// TIA Portal V18 export
// export: Created 2026-03-12T16:04:35.7521041Z, ExportSetting WithDefaults, DisplayName Totally Integrated Automation Portal, DisplayVersion V18 Update 5, DisplayName TIA Portal Openness, DisplayVersion V18 Update 5, DisplayName TIA Portal Version Control Interface, DisplayVersion V18, DisplayName SINAMICS Startdrive Advanced, DisplayVersion V18, DisplayName SINAMICS Startdrive G130, G150, S120, S150, SINAMICS MV, S210, DisplayVersion V18, DisplayName SINAMICS Startdrive G110M, G120, G120C, G120D, G120P, G115D, DisplayVersion V18, DisplayName STEP 7 Professional, DisplayVersion V18 Update 5, DisplayName STEP 7 Safety, DisplayVersion V18, DisplayName WinCC Professional, DisplayVersion V18 Update 5
FUNCTION_BLOCK "FB_MOVE_SKID_DESARENADOR"   // FB33, SCL
{ S7_Optimized_Access := 'TRUE' }
VERSION : 0.1
// stored: AutoNumber true, IsIECCheckEnabled false, IsRetainMemResEnabled false, MemoryReserve 100, SetENOAutomatically false, UDAEnableTagReadback false
   VAR_INPUT
      Dados_Word : Array[10..64] of Int;
      Dados_Bool : Array[0..152] of Bool;
   END_VAR
   VAR_IN_OUT
      SKID_DESARENADOR : Struct
         EMERGENCIA_LIBERADA : Bool;
         AUTOMATICO : Bool;
         MANUAL : Bool;
         POSIÇÃO_INICLA_MANUAL : Bool;
         FLAG_BOMBA_01_LIGADA : Bool;
         FLAG_BOMBA_02_LIGADA : Bool;
         FLAG_SOBRECARGA_DESLOCAMENTO : Bool;
         FLAG_SOBRECARGA_ARRASTADOR01 : Bool;
         FLAG_SOBRECARGA_ARRASTADOR02 : Bool;
         AUXILIAR_ARRASTADOR1_MICRO_CIMA : Bool;
         FLAG_SOBRECARGA_BOMBA01 : Bool;
         FLAG_SOBRECARGA_BOMBA02 : Bool;
         FLAG_DESLOCAMENTO_AVANÇADO : Bool;
         FLAG_DESLOCAMENTO_RECUADO : Bool;
         FLAG_ARRASTADOR01_CIMA : Bool;
         FLAG_ARRASTADOR01_BAIXO : Bool;
         FLAG_ARRASTADOR02_CIMA : Bool;
         FLAG_ARRASTADOR02_BAIXO : Bool;
         DESLOCAMENTO_AVANÇA_IHM : Bool;
         DESLOCAMENTO_MANUAL_AVANÇA : Bool;
         DESLOCAMENTO_RECUA_IHM : Bool;
         DESLOCAMENTO_MANUAL_RECUA : Bool;
         ARRASTADOR01_SOBE_IHM : Bool;
         ARRASTADOR01_SOBE_MANUAL : Bool;
         ARRASTADOR01_DESCE_IHM : Bool;
         ARRASTADOR01_DESCE_MANUAL : Bool;
         ARRASTADOR02_SOBE_IHM : Bool;
         ARRASTADOR02_SOBE_MANUAL : Bool;
         ARRASTADOR02_DESCE_IHM : Bool;
         ARRASTADOR02_DESCE_MANUAL : Bool;
         LIGA_BOMBA01_IHM : Bool;
         LIGA_BOMBA02_IHM : Bool;
         POSICÃO_INICIAL : Bool;
         START_CICLO_IHM : Bool;
         ARRASTADOR01_DESCE_AUTOMATICO : Bool;
         ARRASTADOR02_DESCE_AUTOMATICO : Bool;
         DESLOCAMENTO_AVANÇA_AUTOMATICO : Bool;
         ARRASTADOR01_SOBE_AUTOMATICO : Bool;
         ARRASTADOR02_SOBE_AUTOMATICO : Bool;
         DESLOCAMENTO_RECUA_AUTOMATICO : Bool;
         AUXILIAR_DESLIGA_CICLO : Bool;
         AUXILIAR_DESLIGA_CICLOII : Bool;
         NUMERO_CICLOS_ATINGIDO : Bool;
         CONDIÇÃO_COMPARAÇÃO : Bool;
         NOVO_CICLO_TEMPO : Bool;
         FLAG_NOVO_CICLO : Bool;
         FLAG_ALARME : Bool;
         DESLOCAMENTO_POS_INICIAL : Bool;
         ARRASTADOR01_POS_INICIAL : Bool;
         ARRASTADOR02_POS_INICIAL : Bool;
         BOMBA01_AUTOMATICO : Bool;
         BOMBA02_AUTOMATICO : Bool;
         FLAG_ALARME_IHM : Bool;
         SEGUNDOS_ATINGIDOS : Bool;
         MINUTOS_ATINGIDOS : Bool;
         HORAS_ATINGIDAS : Bool;
         CICLOS_ATUAIS : Int;
         NUMERO_CICLOS_IHM : Int;
         MINUTOS_IHM : Int;
         SEGUNDOS_IHM : Int;
         HORAS_IHM : Int;
         MOVE_SEGUNDOS : Int;
         MOVE_MINUTOS : Int;
         MOVE_HORAS : Int;
      END_STRUCT;
   END_VAR
   // // Dados_Word[10] : Ciclos_Atuais
   // // Dados_Word[20] : Numero_Ciclos_IHM
   // // Dados_Word[30] : Minutos_IHM
   // // Dados_Word[50] : Segundos_IHM
   // // Dados_Word[52] : Horas_IHM
   // // Dados_Word[60] : Move_Segundos
   // // Dados_Word[62] : Move_Minutos
   // // Dados_Word[64] : Move_Horas
   // // Dados_Bool[0] : Emergencia_Liberada
   // // Dados_Bool[1] : Automatico
   // // Dados_Bool[2] : Manual
   // // Dados_Bool[3] : Posição_Inicla_Manual
   // // Dados_Bool[4] : Flag_Bomba_01_Ligada
   // // Dados_Bool[5] : Flag_Bomba_02_Ligada
   // // Dados_Bool[6] : Flag_Sobrecarga_Deslocamento
   // // Dados_Bool[7] : Flag_Sobrecarga_Arrastador01
   // // Dados_Bool[8] : Flag_Sobrecarga_Arrastador02
   // // Dados_Bool[16] : Auxiliar_Arrastador1_Micro_Cima
   // // Dados_Bool[20] : Flag_Sobrecarga_Bomba01
   // // Dados_Bool[21] : Flag_Sobrecarga_Bomba02
   // // Dados_Bool[22] : Flag_Deslocamento_Avançado
   // // Dados_Bool[23] : Flag_Deslocamento_Recuado
   // // Dados_Bool[24] : Flag_Arrastador01_Cima
   // // Dados_Bool[25] : Flag_Arrastador01_Baixo
   // // Dados_Bool[26] : Flag_Arrastador02_Cima
   // // Dados_Bool[27] : Flag_Arrastador02_Baixo
   // // Dados_Bool[40] : Deslocamento_Avança_IHM
   // // Dados_Bool[41] : Deslocamento_Manual_Avança
   // // Dados_Bool[42] : Deslocamento_Recua_IHM
   // // Dados_Bool[43] : Deslocamento_Manual_Recua
   // // Dados_Bool[44] : Arrastador01_Sobe_IHM
   // // Dados_Bool[45] : Arrastador01_Sobe_Manual
   // // Dados_Bool[46] : Arrastador01_Desce_IHM
   // // Dados_Bool[47] : Arrastador01_Desce_Manual
   // // Dados_Bool[48] : Arrastador02_Sobe_IHM
   // // Dados_Bool[49] : Arrastador02_Sobe_Manual
   // // Dados_Bool[50] : Arrastador02_Desce_IHM
   // // Dados_Bool[51] : Arrastador02_Desce_Manual
   // // Dados_Bool[52] : Liga_Bomba01_IHM
   // // Dados_Bool[53] : Liga_Bomba02_IHM
   // // Dados_Bool[54] : Posicão_Inicial
   // // Dados_Bool[55] : Start_Ciclo_IHM
   // // Dados_Bool[56] : Arrastador01_Desce_Automatico
   // // Dados_Bool[57] : Arrastador02_Desce_Automatico
   // // Dados_Bool[58] : Deslocamento_Avança_Automatico
   // // Dados_Bool[59] : Arrastador01_Sobe_Automatico
   // // Dados_Bool[60] : Arrastador02_Sobe_Automatico
   // // Dados_Bool[61] : Deslocamento_Recua_Automatico
   // // Dados_Bool[62] : Auxiliar_Desliga_Ciclo
   // // Dados_Bool[63] : Auxiliar_Desliga_CicloII
   // // Dados_Bool[70] : Numero_Ciclos_Atingido
   // // Dados_Bool[71] : Condição_Comparação
   // // Dados_Bool[75] : Novo_Ciclo_Tempo
   // // Dados_Bool[77] : Flag_Novo_Ciclo
   // // Dados_Bool[80] : Flag_Alarme
   // // Dados_Bool[81] : Deslocamento_Pos_Inicial
   // // Dados_Bool[82] : Arrastador01_Pos_Inicial
   // // Dados_Bool[83] : Arrastador02_Pos_Inicial
   // // Dados_Bool[90] : Bomba01_Automatico
   // // Dados_Bool[91] : Bomba02_Automatico
   // // Dados_Bool[102] : Flag_Alarme_IHM
   // // Dados_Bool[150] : Segundos_Atingidos
   // // Dados_Bool[151] : Minutos_Atingidos
   // // Dados_Bool[152] : Horas_Atingidas
BEGIN
   // ===== BOOL =====
   #SKID_DESARENADOR.EMERGENCIA_LIBERADA := #Dados_Bool[0];
   #SKID_DESARENADOR.AUTOMATICO := #Dados_Bool[1];
   #SKID_DESARENADOR.MANUAL := #Dados_Bool[2];
   #SKID_DESARENADOR.POSIÇÃO_INICLA_MANUAL := #Dados_Bool[3];
   #SKID_DESARENADOR.FLAG_BOMBA_01_LIGADA := #Dados_Bool[4];
   #SKID_DESARENADOR.FLAG_BOMBA_02_LIGADA := #Dados_Bool[5];
   #SKID_DESARENADOR.FLAG_SOBRECARGA_DESLOCAMENTO := #Dados_Bool[6];
   #SKID_DESARENADOR.FLAG_SOBRECARGA_ARRASTADOR01 := #Dados_Bool[7];
   #SKID_DESARENADOR.FLAG_SOBRECARGA_ARRASTADOR02 := #Dados_Bool[8];
   #SKID_DESARENADOR.AUXILIAR_ARRASTADOR1_MICRO_CIMA := #Dados_Bool[16];
   #SKID_DESARENADOR.FLAG_SOBRECARGA_BOMBA01 := #Dados_Bool[20];
   #SKID_DESARENADOR.FLAG_SOBRECARGA_BOMBA02 := #Dados_Bool[21];
   #SKID_DESARENADOR.FLAG_DESLOCAMENTO_AVANÇADO := #Dados_Bool[22];
   #SKID_DESARENADOR.FLAG_DESLOCAMENTO_RECUADO := #Dados_Bool[23];
   #SKID_DESARENADOR.FLAG_ARRASTADOR01_CIMA := #Dados_Bool[24];
   #SKID_DESARENADOR.FLAG_ARRASTADOR01_BAIXO := #Dados_Bool[25];
   #SKID_DESARENADOR.FLAG_ARRASTADOR02_CIMA := #Dados_Bool[26];
   #SKID_DESARENADOR.FLAG_ARRASTADOR02_BAIXO := #Dados_Bool[27];

   #SKID_DESARENADOR.DESLOCAMENTO_AVANÇA_IHM := #Dados_Bool[40];
   #SKID_DESARENADOR.DESLOCAMENTO_MANUAL_AVANÇA := #Dados_Bool[41];
   #SKID_DESARENADOR.DESLOCAMENTO_RECUA_IHM := #Dados_Bool[42];
   #SKID_DESARENADOR.DESLOCAMENTO_MANUAL_RECUA := #Dados_Bool[43];

   #SKID_DESARENADOR.ARRASTADOR01_SOBE_IHM := #Dados_Bool[44];
   #SKID_DESARENADOR.ARRASTADOR01_SOBE_MANUAL := #Dados_Bool[45];
   #SKID_DESARENADOR.ARRASTADOR01_DESCE_IHM := #Dados_Bool[46];
   #SKID_DESARENADOR.ARRASTADOR01_DESCE_MANUAL := #Dados_Bool[47];

   #SKID_DESARENADOR.ARRASTADOR02_SOBE_IHM := #Dados_Bool[48];
   #SKID_DESARENADOR.ARRASTADOR02_SOBE_MANUAL := #Dados_Bool[49];
   #SKID_DESARENADOR.ARRASTADOR02_DESCE_IHM := #Dados_Bool[50];
   #SKID_DESARENADOR.ARRASTADOR02_DESCE_MANUAL := #Dados_Bool[51];

   #SKID_DESARENADOR.LIGA_BOMBA01_IHM := #Dados_Bool[52];
   #SKID_DESARENADOR.LIGA_BOMBA02_IHM := #Dados_Bool[53];
   #SKID_DESARENADOR.POSICÃO_INICIAL := #Dados_Bool[54];
   #SKID_DESARENADOR.START_CICLO_IHM := #Dados_Bool[55];

   #SKID_DESARENADOR.ARRASTADOR01_DESCE_AUTOMATICO := #Dados_Bool[56];
   #SKID_DESARENADOR.ARRASTADOR02_DESCE_AUTOMATICO := #Dados_Bool[57];
   #SKID_DESARENADOR.DESLOCAMENTO_AVANÇA_AUTOMATICO := #Dados_Bool[58];
   #SKID_DESARENADOR.ARRASTADOR01_SOBE_AUTOMATICO := #Dados_Bool[59];
   #SKID_DESARENADOR.ARRASTADOR02_SOBE_AUTOMATICO := #Dados_Bool[60];
   #SKID_DESARENADOR.DESLOCAMENTO_RECUA_AUTOMATICO := #Dados_Bool[61];

   #SKID_DESARENADOR.AUXILIAR_DESLIGA_CICLO := #Dados_Bool[62];
   #SKID_DESARENADOR.AUXILIAR_DESLIGA_CICLOII := #Dados_Bool[63];

   #SKID_DESARENADOR.NUMERO_CICLOS_ATINGIDO := #Dados_Bool[70];
   #SKID_DESARENADOR.CONDIÇÃO_COMPARAÇÃO := #Dados_Bool[71];
   #SKID_DESARENADOR.NOVO_CICLO_TEMPO := #Dados_Bool[75];
   #SKID_DESARENADOR.FLAG_NOVO_CICLO := #Dados_Bool[77];
   #SKID_DESARENADOR.FLAG_ALARME := #Dados_Bool[80];

   #SKID_DESARENADOR.DESLOCAMENTO_POS_INICIAL := #Dados_Bool[81];
   #SKID_DESARENADOR.ARRASTADOR01_POS_INICIAL := #Dados_Bool[82];
   #SKID_DESARENADOR.ARRASTADOR02_POS_INICIAL := #Dados_Bool[83];

   #SKID_DESARENADOR.BOMBA01_AUTOMATICO := #Dados_Bool[90];
   #SKID_DESARENADOR.BOMBA02_AUTOMATICO := #Dados_Bool[91];

   #SKID_DESARENADOR.FLAG_ALARME_IHM := #Dados_Bool[102];
   #SKID_DESARENADOR.SEGUNDOS_ATINGIDOS := #Dados_Bool[150];
   #SKID_DESARENADOR.MINUTOS_ATINGIDOS := #Dados_Bool[151];
   #SKID_DESARENADOR.HORAS_ATINGIDAS := #Dados_Bool[152];


   // ===== INT =====
   #SKID_DESARENADOR.CICLOS_ATUAIS := #Dados_Word[10];
   #SKID_DESARENADOR.NUMERO_CICLOS_IHM := #Dados_Word[20];
   #SKID_DESARENADOR.MINUTOS_IHM := #Dados_Word[30];
   #SKID_DESARENADOR.SEGUNDOS_IHM := #Dados_Word[50];
   #SKID_DESARENADOR.HORAS_IHM := #Dados_Word[52];
   #SKID_DESARENADOR.MOVE_SEGUNDOS := #Dados_Word[60];
   #SKID_DESARENADOR.MOVE_MINUTOS := #Dados_Word[62];
   #SKID_DESARENADOR.MOVE_HORAS := #Dados_Word[64];
END_FUNCTION_BLOCK
